# EPICS StreamDevice protocol: TEST/TEST-IOC-01App/protocol/test.proto
Terminator = LF;

writeString {
    out "%s";
}

readString {
    in "%s";
}
